{attribute 'qualified_only'}
{attribute 'strict'}
TYPE E_DALIExtendedFadeTime :
(
	NoFade := 0,
	onehundred := 1,
	twohundred := 2,
	threehundred := 3,
	fourhundred := 4,
	fivehundred := 5,
	sixhundred := 6,
	sevenhundred := 7,
	eighthundred := 8,
	ninehundred := 9,
	onethousand := 10,
	onethousandonehundred := 11,
	onethousandtwohundred := 12,
	onethousandthreehundred := 13,
	onethousandfourhundred := 14,
	onethousandfivehundred := 15,
	onethousandsixhundred	:= 16,
	onesecond := 17,
	twoseconds := 18,
	threeseconds := 19,
	fourseconds := 20,
	fiveseconds := 21,
	sixseconds := 22,
	sevenseconds := 23,
	eightseconds := 24,
	nineseconds := 25,
	tenseconds := 26,
	elevenseconds := 27,
	twelveseconds := 28,
	thirteenseconds := 29,
	fourteenseconds := 30,
	fifteenseconds := 31,
	sixteenseconds := 32,
	ten1seconds := 33,
	twentyseconds := 34,
	thirtyseconds := 35,
	fourtyseconds := 36,
	fiftyseconds := 37,
	sixtyseconds := 38,
	seventyseconds := 39,
	eightyseconds := 40,
	ninetyseconds := 41,
	onehundredseconds := 42,
	onehundredtenseconds := 43,
	onehundredtwentyseconds := 44,
	onehundredthirtyseconds := 45,
	onehundredfourtyseconds := 46,
	onehundredfiftyseconds := 47,
	onehundredsixtyseconds := 48,
	oneminute := 49,
	twominutes := 50,
	threeminutes := 51,
	fourminutes := 52,
	fiveminutes := 53,
	sixminutes := 54,
	sevenminutes := 55,
	eightminutes := 56,
	nineminutes := 57,
	tenminutes := 58,
	elevenminutes := 59,
	twelveminutes := 60,
	thirteenminutes := 61,
	fourteenminutes := 62,
	fifteenminutes := 63,
	sixteenminutes := 64,
	unknown := 255
);
END_TYPE

(* stored: Version 1.1.0.1, ProductVersion 3.1.4024.10
   EnumerationTextList E_DALIExtendedFadeTime: Id {ac38bbfc-184c-4046-930a-6ec149e0c74c} *)
